// TwinCAT 3 PLC project FileDownload
// ProgramVersion: 3.1.0.5
// libraries:
//   Tc2_FTP,newest,Beckhoff Automation GmbH
//   Tc2_Standard,newest,Beckhoff Automation GmbH
//   Tc2_System,newest,Beckhoff Automation GmbH
//   Tc3_Module,newest,Beckhoff Automation GmbH
// project tree:
//   / PlcTask.TcTTO
//   POUs/ MAIN.TcPOU
// (motion and I/O tree: see PLC project fileupload)
// real-time tasks:
//   TASK PlcTask: cycle T#10ms, priority 20, ADS port 350

CONFIGURATION FileDownload
    RESOURCE PLC ON TwinCAT3
        TASK PlcTask(INTERVAL := T#10ms, PRIORITY := 20);
        PROGRAM MAIN WITH PlcTask : MAIN;
    END_RESOURCE
END_CONFIGURATION

// ---- POUs/MAIN.TcPOU
PROGRAM MAIN
VAR
	RisingEdge 			: R_TRIG;
	startstop 			: BOOL;
	state				: BYTE;
	FB_FTP_Open1 		: FB_FTP_Open;
	FB_FTP_FileDownload1: FB_FTP_FileDownload;
	FB_FTP_Close1 		: FB_FTP_Close;
	busy 				: BOOL;
	err 				: BOOL;
	errid 				: UDINT;
	handle 				: T_HFTP;
	progress 			: UDINT;
END_VAR

RisingEdge(CLK:= startstop);
IF RisingEdge.Q THEN
	state := 1;
END_IF

CASE state OF
	0:
		;

	1:
		FB_FTP_Open1(
			sNetID:= ,
			sHost:= '172.17.216.47',
			nPort:= 21,
			sUsername:= 'TestUser',
			sPassword:= 'TestPwd123',
			bExecute:= TRUE,
			tTimeout:= T#15s,
			bBusy=> busy,
			bError=> err,
			nErrId=> errid,
			hFTP=> handle);

		IF NOT busy AND NOT err THEN
			FB_FTP_Open1(bExecute:= FALSE);
			state := 2;
		END_IF

	2:
		FB_FTP_FileDownload1(
			sNetID:= ,
			hFTP:= handle,
			sSrcFile:= '\TestFolder\File1.txt',
			sDesFile:= '\Program Files\TestFile1.txt',
			bExecute:= TRUE,
			tTimeout:= T#15s,
			bBusy => busy,
			bError => err,
			nErrId => errid,
			nProgress => progress);

		IF NOT busy AND NOT err THEN
			FB_FTP_FileDownload1(bExecute:= FALSE);
			state := 3;
		END_IF

	3:
		FB_FTP_Close1(
			sNetID:= ,
			hFTP:= handle,
			bExecute:= TRUE,
			tTimeout:= T#15s,
			bBusy => busy,
			bError => err,
			nErrId => errid);

		IF NOT busy AND NOT err THEN
			FB_FTP_Close1(bExecute:= FALSE);
			state := 0;
		END_IF

END_CASE

END_PROGRAM
